// Mitsubishi GX Works2 project: n08   PLC: Q02/Q02H

PROGRAM MAIN
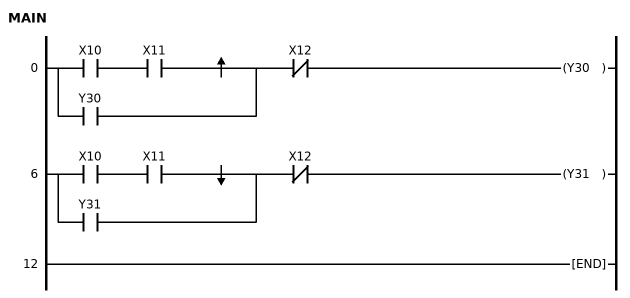
0     LD      X10
      AND     X11
      MEP
      OR      Y30
      ANI     X12
      OUT     Y30
6     LD      X10
      AND     X11
      MEF
      OR      Y31
      ANI     X12
      OUT     Y31
12    END
END_PROGRAM
